TYPE ST_System_BSp_KueW_Stellwert :
STRUCT
	Anford_Aussenfassadenaktivierung	: BOOL;
	Anford_Pumpe						: BOOL;
	Einschaltperiode_Max				: TIME := T#5S;
	Einschalten							: BOOL;
END_STRUCT
END_TYPE

(* stored: Version 1.1.0.1, ProductVersion 3.1.4024.9
   DUT ST_System_BSp_KueW_Stellwert: Id {9e17fcc6-9890-466d-97b4-06de2cec4111} *)
